TYPE SAdsSymbol :
STRUCT
	IsSet: BOOL;		// indicates whether this target is defined
	DataType: EDataType;
	
	NetId: T_AmsNetID;	// alias for STRING(23)
	Port: T_AmsPort;	// alias for UINT
	
	IdxGrp: UDINT;
	IdxOffs: UDINT;
END_STRUCT
END_TYPE

(* stored: Version 1.1.0.1
   DUT SAdsSymbol: Id {b359cdc7-dae0-4a1f-9c17-a9a848f77eba} *)
